// TIA Portal V20 export
// export: Created 2025-12-01T14:57:09.8220942Z, ExportSetting None, DisplayName Totally Integrated Automation Portal, DisplayVersion V20 Update 3, DisplayName TIA Portal Openness, DisplayVersion V20 Update 3, DisplayName TIA Portal Version Control Interface, DisplayVersion V20 Update 3, DisplayName STEP 7 Professional, DisplayVersion V20 Update 3, DisplayName STEP 7 Safety, DisplayVersion V20 Update 2, DisplayName WinCC Basic/Comfort/Advanced, DisplayVersion V20 Update 3, DisplayName WinCC Professional, DisplayVersion V20 Update 3, DisplayName WinCC Unified, DisplayVersion V20 Update 3
FUNCTION "FC729_ResetearMesa" : Void   // FC729, LAD
{ S7_Optimized_Access := 'FALSE' }
AUTHOR : TRACKING
NAME : 20130301
VERSION : 3.0
// stored: AutoNumber false, SetENOAutomatically false
   VAR_INPUT
      NumMesa : UInt;   // Numero de Mesa a Resetear
      SinPresencia : Bool;   // Reset Manual, en Mesa sin Presencia
   END_VAR
   VAR_TEMP
      Mesa : UInt;
      NumeroUT : UInt;
      ValorReturn : Int;
      Cero : Byte;
      ResetTotal : Bool;
      ResetParcial : Bool;
   END_VAR
BEGIN

NETWORK
TITLE = Inicializar
///////////////////////////////////////////////////////////////////////////////
///////////////////////////////////////////////////////////////////////////////
///////////////////////////////////////////////////////////////////////////////
// --- Inicializar

      L     #NumMesa;  // Pasar a Temporal
      T     #Mesa;

      SET;
      R     #ResetTotal;  // Reseteo las variables de tipo
      R     #ResetParcial;




NETWORK
TITLE = Resteo de las variables de la Mesa en la BD
///////////////////////////////////////////////////////////////////////////////
///////////////////////////////////////////////////////////////////////////////
///////////////////////////////////////////////////////////////////////////////
// --- Reset en la Cola de la Mesa
// --- * Desactivar todos los protocolos de la Mesa
// --- * Desactivar las los bits enviados al Vehiculo inteligente

      L     0;  // Limpieza de los Protocolos
      T     "DB810_ColasMesas".Colas[#Mesa].EstadoOrdenMesa;
      T     "DB810_ColasMesas".Colas[#Mesa].EstadoPresenciaMesa;

      L     0;  // Limpieza de las Comunicaciones
      T     #Cero;
      CALL  FILL
      ( BVAL    := #Cero,
        RET_VAL := #ValorReturn,
        BLK     := "DB841_Recepcion".Mesa[#Mesa]
      );



NETWORK
TITLE = Distribuir Segun el Tipo de Reset Total o Parcial
///////////////////////////////////////////////////////////////////////////////
///////////////////////////////////////////////////////////////////////////////
///////////////////////////////////////////////////////////////////////////////
// --- Recoger el Tipo de Reset del Dispositivo Mesa
      SET;  // Bit de ResetTotal
      A     "DB831_Mesas".Mesas[#Mesa].Memorias.M_ResetTotal;
      S     #ResetTotal;

      SET;  // Bit de ResetParcial
      A     "DB831_Mesas".Mesas[#Mesa].Memorias.M_ResetParcial;
      S     #ResetParcial;


// --- Distribuir segun tipo de Reset
      SET;
      A     #ResetTotal;
      JC    ResetTotal_EnMesa;  // Es Reset Total ?
      JU    ResetParcial_EnMesa;  // Sino Reset Parcial



NETWORK
TITLE = Reset Total de Mesa
///////////////////////////////////////////////////////////////////////////////
///////////////////////////////////////////////////////////////////////////////
///////////////////////////////////////////////////////////////////////////////
// ---     RESET TOTAL --> Borrado de todas las UT's de la Mesa
// ---
// --- * Recorrer las UT's de la Mesa
// ---   + Eliminacion de la UT

ResetTotal_EnMesa:NOP   0;
      L     "DB810_ColasMesas".Colas[#Mesa].UT_PrimeraMesa;
      T     #NumeroUT;


///////////////////////////////////////////////////////////////////////////////
///////////////////////////////////////////////////////////////////////////////
BucleResetTotal_EnMesa:NOP   0;
      L     #NumeroUT;
      L     0;
      ==I;  // No hay más UT's
      JC    Final_Funcion;

      CALL  "FC722_EliminarUT_DeMesa"
      ( NumeroUT := #NumeroUT
      );

      L     "DB810_ColasMesas".Colas[#Mesa].UT_PrimeraMesa;
      T     #NumeroUT;

      JU    BucleResetTotal_EnMesa;



NETWORK
TITLE = Reset Parcial de Mesa
///////////////////////////////////////////////////////////////////////////////
///////////////////////////////////////////////////////////////////////////////
///////////////////////////////////////////////////////////////////////////////
// ---     RESET PARCIAL --> Reset en los datos de las UT's
// ---
// --- * Recorrer las UT's de la Mesa
// ---   + Poner el codigo de reset en EmisionUT o RecepcionUT
// ---   + Limpiar el resto

ResetParcial_EnMesa:NOP   0;
      L     "DB810_ColasMesas".Colas[#Mesa].UT_PrimeraMesa;
      T     #NumeroUT;


///////////////////////////////////////////////////////////////////////////////
///////////////////////////////////////////////////////////////////////////////
BucleResetParcial_EnMesa:NOP   0;
      L     #NumeroUT;
      L     0;
      ==I;
      JC    Final_Funcion;  // No hay más UT's


///////////////////////////////////////////////////////////////////////////////
// --- Ver que Tipo de Mesa (Con o Sin Presencia en el Reset)

      A     #SinPresencia;
      O     "DB850_DefinicionMesas".Mesa[#Mesa].ConfigMesa.SinPresenciaEnReset;
      JC    ResetParcial_SinPresencia;  // Mesa Sin Presencia ??
      JU    ResetParcial_ConPresencia;  // Mesa Con Presencia ??


///////////////////////////////////////////////////////////////////////////////
///////////////////////////////////////////////////////////////////////////////
// --- Mesa Con Pressencia
ResetParcial_ConPresencia:NOP   0;
      L     0;
      T     "DB812_UTs_Control".UT[#NumeroUT].EstadoEmisionUT;
      T     "DB812_UTs_Control".UT[#NumeroUT].EstadoRecepcionUT;
//      T     "DB815_DatosUT".Datos_UTs[#NumeroUT].EstadoGeneralUT // ????
      T     "DB812_UTs_Control".UT[#NumeroUT].EstadoEventoRecibido;
      T     "DB812_UTs_Control".UT[#NumeroUT].EstadoEventoAGenerar;

      L     13;
      T     "DB812_UTs_Control".UT[#NumeroUT].EstadoEmisionUT;

// Continuar con la Siguiente UT
      L     "DB812_UTs_Control".UT[#NumeroUT].UT_SiguienteMesa;
      T     #NumeroUT;

      JU    BucleResetParcial_EnMesa;


///////////////////////////////////////////////////////////////////////////////
///////////////////////////////////////////////////////////////////////////////
// --- Mesa Sin Pressencia
ResetParcial_SinPresencia:NOP   0;
      L     0;
      T     "DB812_UTs_Control".UT[#NumeroUT].EstadoEmisionUT;
      T     "DB812_UTs_Control".UT[#NumeroUT].EstadoRecepcionUT;
//      T     "DB815_DatosUT".Datos_UTs[#NumeroUT].EstadoGeneralUT // ????
      T     "DB812_UTs_Control".UT[#NumeroUT].EstadoEventoRecibido;
      T     "DB812_UTs_Control".UT[#NumeroUT].EstadoEventoAGenerar;

      L     13;
      T     "DB812_UTs_Control".UT[#NumeroUT].EstadoRecepcionUT;

// Continuar con la Siguiente UT
      L     "DB812_UTs_Control".UT[#NumeroUT].UT_SiguienteMesa;
      T     #NumeroUT;

      JU    BucleResetParcial_EnMesa;



NETWORK
TITLE = Final de la Funcion
///////////////////////////////////////////////////////////////////////////////
///////////////////////////////////////////////////////////////////////////////
///////////////////////////////////////////////////////////////////////////////
// --- FINAL DE LA FUNCION

Final_Funcion:NOP   0;


END_FUNCTION
